ABB RobotStudio station: Simuleringsopgave_2_20200505-151904.rsstn

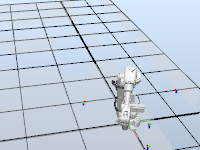
Station Simuleringsopgave_2 (saved by RobotStudio 7.0.8746.631)
Controller IRB_2600_20kg_1.65m_1
  mechanical unit ROB_1: IRB2600_20_165__02, 6 joints, base frame (0, 0, 0) mm
Layout (positions relative to the parent item):
  - IRB2600_20_165__02 [mechanism, from Robots\IRB2600_20_165_G_02.rslib] at (0, 0, 0) mm; joint values [-0.4129, 0.1779, 0.5307, -6.2924, 0.8625, 6.3308] (rad or m)
  - MyNewTool [mechanism] at (872.04, -382.72, 618.96) mm, rotated rx -179.6 ry 0 rz 153.96 deg
      TCP MyNewTool at (0, 0, 30) mm
      links: SimpleGripper
  - Sorter_kassser_COLLADA_EXPORT [graphiccomponentgroup]
    - Assemblies [graphiccomponentgroup]
      - Section1 [graphiccomponentgroup]
        - ABB_IRC5_ctrl [graphiccomponentgroup]
          - ABB_IRC5_ctrl_1 [graphiccomponentgroup]
            - Mesh0 [part]
        - Beacon [graphiccomponentgroup]
          - BEACON1 [graphiccomponentgroup]
            - Mesh1 [part]
            - Mesh2 [part]
            - Mesh3 [part]
            - Mesh4 [part]
            - Mesh5 [part]
            - Mesh6 [part]
            - Mesh7 [part]
            - Mesh8 [part]
            - Mesh9 [part]
            - Mesh10 [part]
        - Conveyor__Straight_ [graphiccomponentgroup]
          - CONVEYOR1 [graphiccomponentgroup]
            - Mesh11 [part]
            - Mesh12 [part]
            - Mesh13 [part]
            - Mesh14 [part]
          - CONVEYOR2 [graphiccomponentgroup]
            - Mesh15 [part]
            - Mesh16 [part]
            - Mesh17 [part]
          - CONVEYOR3 [graphiccomponentgroup]
            - Mesh18 [part]
            - Mesh19 [part]
            - Mesh20 [part]
            - Mesh21 [part]
            - Mesh22 [part]
          - CONVEYOR4 [graphiccomponentgroup]
            - Mesh23 [part]
            - Mesh24 [part]
            - Mesh25 [part]
          - CONVEYOR5 [graphiccomponentgroup]
            - Mesh26 [part]
            - Mesh27 [part]
            - Mesh28 [part]
          - CONVEYOR6 [graphiccomponentgroup]
            - Mesh29 [part]
            - Mesh30 [part]
            - Mesh31 [part]
            - Mesh32 [part]
            - Mesh33 [part]
          - CONVEYOR7 [graphiccomponentgroup]
            - Mesh34 [part]
            - Mesh35 [part]
            - Mesh36 [part]
          - CONVEYOR8 [graphiccomponentgroup]
            - Mesh37 [part]
            - Mesh38 [part]
            - Mesh39 [part]
          - CONVEYOR9 [graphiccomponentgroup]
            - Mesh40 [part]
            - Mesh41 [part]
            - Mesh42 [part]
        - Cube [graphiccomponentgroup]
          - Cube1 [graphiccomponentgroup]
            - Mesh43 [part]
            - Mesh44 [part]
            - Mesh45 [part]
            - Mesh46 [part]
            - Mesh47 [part]
        - Eater [graphiccomponentgroup]
          - EATER1 [graphiccomponentgroup]
            - Mesh48 [part]
          - EATER2 [graphiccomponentgroup]
            - Mesh49 [part]
          - EATER3 [graphiccomponentgroup]
            - Mesh50 [part]
        - Display [graphiccomponentgroup]
          - EaterLarge [graphiccomponentgroup]
            - Mesh51 [part]
            - Mesh52 [part]
            - Mesh53 [part]
            - Mesh54 [part]
            - Mesh55 [part]
            - Mesh56 [part]
            - Mesh57 [part]
            - Mesh58 [part]
            - Mesh59 [part]
            - Mesh60 [part]
            - Mesh61 [part]
          - EaterMedium [graphiccomponentgroup]
            - Mesh62 [part]
            - Mesh63 [part]
            - Mesh64 [part]
            - Mesh65 [part]
            - Mesh66 [part]
            - Mesh67 [part]
            - Mesh68 [part]
            - Mesh69 [part]
            - Mesh70 [part]
            - Mesh71 [part]
            - Mesh72 [part]
          - EaterSmall [graphiccomponentgroup]
            - Mesh73 [part]
            - Mesh74 [part]
            - Mesh75 [part]
            - Mesh76 [part]
            - Mesh77 [part]
            - Mesh78 [part]
            - Mesh79 [part]
            - Mesh80 [part]
            - Mesh81 [part]
            - Mesh82 [part]
            - Mesh83 [part]
        - Fences [graphiccomponentgroup]
          - FENCE1 [graphiccomponentgroup]
            - Mesh84 [part]
            - Mesh85 [part]
            - Mesh86 [part]
            - Mesh87 [part]
            - Mesh88 [part]
            - Mesh89 [part]
            - Mesh90 [part]
            - Mesh91 [part]
            - Mesh92 [part]
            - Mesh93 [part]
          - FENCE4 [graphiccomponentgroup]
            - Mesh94 [part]
            - Mesh95 [part]
            - Mesh96 [part]
            - Mesh97 [part]
            - Mesh98 [part]
            - Mesh99 [part]
            - Mesh100 [part]
            - Mesh101 [part]
            - Mesh102 [part]
            - Mesh103 [part]
          - FENCE5 [graphiccomponentgroup]
            - Mesh104 [part]
            - Mesh105 [part]
            - Mesh106 [part]
            - Mesh107 [part]
            - Mesh108 [part]
            - Mesh109 [part]
            - Mesh110 [part]
            - Mesh111 [part]
            - Mesh112 [part]
            - Mesh113 [part]
        - Scale [graphiccomponentgroup]
          - Scale_Weight [graphiccomponentgroup]
            - Mesh114 [part]
            - Mesh115 [part]
            - Mesh116 [part]
            - Mesh117 [part]
        - Text [graphiccomponentgroup]
          - Text1 [graphiccomponentgroup]
            - Mesh118 [part]
          - Text2 [graphiccomponentgroup]
            - Mesh119 [part]
          - Text3 [graphiccomponentgroup]
            - Mesh120 [part]
    - Motors [graphiccomponentgroup]
      - Surface [graphiccomponentgroup]
        - MOTOR1 [graphiccomponentgroup]
          - Mesh121 [part]
          - Mesh122 [part]
          - Mesh123 [part]
          - Mesh124 [part]
          - Mesh125 [part]
        - MOTOR2 [graphiccomponentgroup]
          - Mesh126 [part]
          - Mesh127 [part]
        - MOTOR3 [graphiccomponentgroup]
          - Mesh128 [part]
          - Mesh129 [part]
Attachment: IRB2600_20_165__02 is attached to Cube1
Attachment: MyNewTool is attached to IRB2600_20_165__02 / Link6
Targets, tools, work objects and paths stored in the station, written as RAPID:
! task T_ROB1
MODULE CalibData
  TASK PERS wobjdata Workobject_1:=[FALSE,TRUE,"",[[0,0,0],[1,0,0,0]],[[0,0,0],[1,0,0,0]]];
  PERS tooldata MyNewTool:=[TRUE,[[0,0,30],[1,0,0,0]],[1,[0,0,1],[1,0,0,0],0,0,0]];
ENDMODULE

! task T_ROB1
MODULE Module1
  CONST robtarget PicKUp:=[[996.139868276,-0.000086478,170.226118879],[0.000036866,0.000002225,0.999993783,-0.00352606],[0,-5,4,0],[9E+09,9E+09,9E+09,9E+09,9E+09,9E+09]];
  CONST robtarget Home:=[[996.139869233,-0.000090103,615.626718052],[0.000036871,0.000002267,0.999993783,-0.003526076],[0,-5,4,0],[9E+09,9E+09,9E+09,9E+09,9E+09,9E+09]];
  CONST robtarget Small:=[[6.065699913,-908.240962462,615.626905136],[0.002646356,-0.757323123,-0.653030822,0.002330353],[-1,-5,4,0],[9E+09,9E+09,9E+09,9E+09,9E+09,9E+09]];
  CONST robtarget Big:=[[-3.693582301,939.352796807,615.626909553],[0.002655413,-0.746102912,0.665821305,-0.002320143],[1,-5,3,0],[9E+09,9E+09,9E+09,9E+09,9E+09,9E+09]];
ENDMODULE

